# EPICS StreamDevice protocol: iocBoot/ioc13test/testIPServer.proto
InTerminator = CR LF;
OutTerminator = CR LF;
read {
    in "%#s";
}

write {
    out "%s";
}
